// TIA Portal V18 export
ORGANIZATION_BLOCK "03_CYC_INT2"   // OB32, LAD, CyclicInterrupt
TITLE = "Cyclic Interrupt"
{ S7_Optimized_Access := 'FALSE' }
// stored: AutoNumber false, SetENOAutomatically false
   VAR_TEMP
      OB32_EV_CLASS : Byte;   // Bits 0-3 = 1 (Coming event), Bits 4-7 = 1 (Event class 1)
      OB32_STRT_INF : Byte;   // 16#33 (OB 32 has started)
      OB32_PRIORITY : Byte;   // Priority of OB Execution
      OB32_OB_NUMBR : Byte;   // 32 (Organization block 32, OB32)
      OB32_RESERVED_1 : Byte;   // Reserved for system
      OB32_RESERVED_2 : Byte;   // Reserved for system
      OB32_PHS_OFFSET : Int;   // Phase offset (integer, milliseconds)
      OB32_RESERVED_3 : Int;   // Reserved for system
      OB32_EXC_FREQ : Int;   // Frequency of execution (msec)
      OB32_DATE_TIME : Date_And_Time;   // Date and time OB32 started
   END_VAR
BEGIN

REGION Network 1
   // //Keep resource code
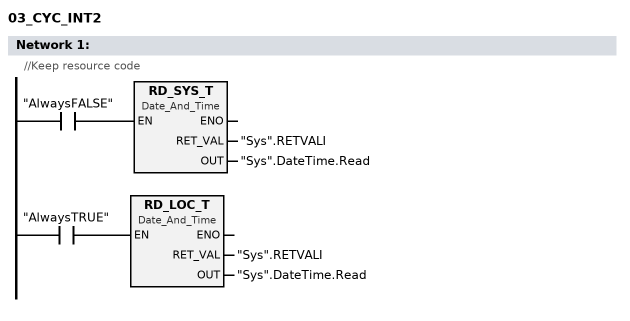
   RUNG wire#powerrail
      Contact( "AlwaysFALSE" )
      { S7_Templates := "date_type := Date_And_Time" } RD_SYS_T(RET_VAL => "Sys".RETVALI, OUT => "Sys".DateTime.Read)
   END_RUNG
   RUNG wire#powerrail
      Contact( "AlwaysTRUE" )
      { S7_Templates := "date_type := Date_And_Time" } RD_LOC_T(RET_VAL => "Sys".RETVALI, OUT => "Sys".DateTime.Read)
   END_RUNG
   // the same network as SCL:
   IF "AlwaysFALSE" THEN "Sys".RETVALI := RD_SYS_T(OUT => "Sys".DateTime.Read); END_IF;
   IF "AlwaysTRUE" THEN "Sys".RETVALI := RD_LOC_T(OUT => "Sys".DateTime.Read); END_IF;
END_REGION

NETWORK
TITLE = Diagnostic
//      CALL  "Diagnostic"
//         iCPUType :=2
//         iDBNum   :=3001
//         iOffset  :=0


END_ORGANIZATION_BLOCK
